// TIA Portal V19 export
VAR_GLOBAL   // PLC tag table "U2Em1_Input"
   trayAutomaticDischargeDetectionU2Em1 AT %I170.1 : Bool;   // Em80_拘束滚筒托盘出料检测
   trayAutomaticFeedingDetectionU2Em1 AT %I170.0 : Bool;   // Em80_拘束滚筒托盘入料检测
   restraintTrayAntiReverseDetection2U2Em1 AT %I174.5 : Bool;   // Em80_拘束托盘防反检测_2
   restraintTrayAntiReverseDetection1U2Em1 AT %I174.4 : Bool;   // Em80_拘束托盘防反检测_1
END_VAR
